RoboDK station: welding.rdk

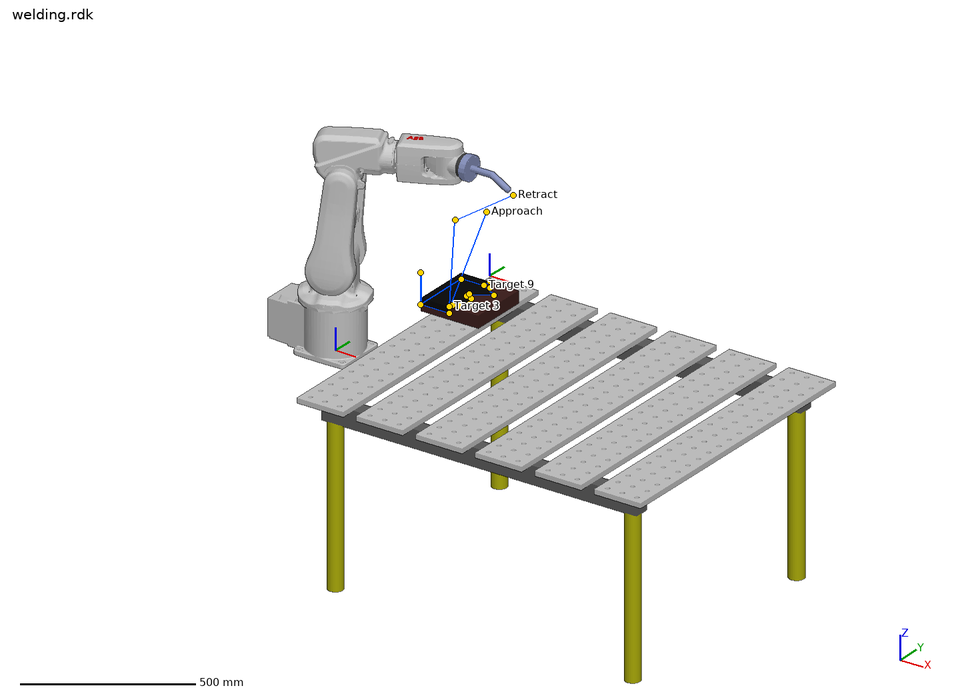
[picture v0: the station drawn from its stored meshes, robots at their saved joint values, targets as dots, program paths as lines]
Station welding (saved by RoboDK 5.3.4). Poses are relative to the parent item; angles as X-Y-Z fixed-axis rotations.
  - frame ABB IRB 120-3/0.6 Base at (0, 0, 0) mm
    - robot ABB IRB 120-3/0.6: 6 axes, payload 3 kg, reach 580 mm, repeatability 0.01 mm, weight 25 kg
        modified DH rows (alpha deg, a mm, theta deg, d mm): 0, 0, 0, 290; -90, 0, -90, 0; 0, 270, 0, 0; -90, 70, 0, 302; 90, 0, 0, 0; -90, 0, 180, 72
        joint limits [-165, -110, -90, -160, -120, -400] to [165, 110, 70, 160, 120, 400]; home [0, 0, 0, 0, 0, 0]; saved at [23.746, 6.012, -6.294, -89.359, 23.748, 89.3]
      - tool AssemblyWeldingTorch, TCP at (45, 0, 150) mm, rotated rx 0 ry 30 rz 0 deg, size 80 x 153.6 x 80.2 mm, geometry from AssemblyWeldingTorch.STEP
  - object Table at (800, 0, 100) mm, size 1193.8 x 965.2 x 609.6 mm, geometry from welding_table.sld
  - frame worktable at (200, 480, 100) mm
    - object Task1_Part2 at (180, -600, 200) mm, rotated rx 90 ry 0 rz 0 deg, size 160 x 20 x 200 mm, geometry from Task1_Part2.STEP
    - object Task1_Part1 at (280, -600, 200) mm, rotated rx 90 ry 0 rz 0 deg, size 200 x 40 x 200 mm, geometry from Task1_Part1.STEP
    - target Approach (Cartesian target) at (324, -480, 485) mm, rotated rx -180 ry 60 rz -180 deg; joints [0, 0, 0, 0, 0, 0] of ABB IRB 120-3/0.6
    - target Target 3 (Cartesian target) at (280, -600, 220) mm, rotated rx -180 ry 30 rz 180 deg; joints [-21.146, 7.513, 21.973, -96.878, -18.342, 86.297] of ABB IRB 120-3/0.6
    - target Target 4 (Cartesian target) at (280, -585, 220) mm, rotated rx -177.69 ry 30 rz 179.62 deg; joints [-17.055, 5.876, 23.812, 85.17, 12.458, -94.648] of ABB IRB 120-3/0.6
    - target Target 6 (Cartesian target) at (280, -515, 220) mm, rotated rx -177.69 ry 30 rz -175.38 deg; joints [-7.356, 3.4, 26.47, 86.971, 8.377, -94.106] of ABB IRB 120-3/0.6
    - target Target 7 (Cartesian target) at (280, -500, 220) mm, rotated rx -177.69 ry 20 rz -175.38 deg; joints [-3.841, 7.541, 16.793, 16.097, 16.374, -22.068] of ABB IRB 120-3/0.6
    - target Target 8 (Cartesian target) at (340, -465, 220) mm, rotated rx -177.69 ry 20 rz -175.38 deg; joints [1.761, 20.013, 1.699, 0.611, 18.24, -3.567] of ABB IRB 120-3/0.6
    - target Target 9 (Cartesian target) at (280, -430, 220) mm, rotated rx -177.69 ry 20 rz -175.38 deg; joints [7.944, 8.066, 16.204, -16.244, 16.455, 16.603] of ABB IRB 120-3/0.6
    - target Target 10 (Cartesian target) at (280, -400, 220) mm, rotated rx -177.69 ry 30 rz -175.38 deg; joints [13.586, 4.724, 25.061, -86.161, 9.774, 89.486] of ABB IRB 120-3/0.6
    - target Target 10-11 turning (Cartesian target) at (280, -400, 220) mm, rotated rx -90 ry 0 rz -150 deg; joints [36.548, 32.886, 19.556, 71.022, -75.96, 234.799] of ABB IRB 120-3/0.6
    - target Target 11 (Cartesian target) at (280, -400, 200) mm, rotated rx -90 ry 0 rz -150 deg; joints [36.548, 35.685, 19.831, 70.324, -76.978, -122.216] of ABB IRB 120-3/0.6
    - target Target 12 (Cartesian target) at (180, -400, 200) mm, rotated rx -90 ry 0 rz -150 deg; joints [47.566, 24.233, 38.454, -101.084, 84.33, 63.237] of ABB IRB 120-3/0.6
    - target Target 12-13 turning (Cartesian target) at (180, -400, 200) mm, rotated rx -90 ry 0 rz -60 deg; joints [-21.316, 14.165, 53.197, -81.976, -86.668, -67.596] of ABB IRB 120-3/0.6
    - target Target 13 (Cartesian target) at (180, -600, 200) mm, rotated rx -90 ry 0 rz -60 deg; joints [-51.555, 33.15, 24.081, -108.374, -101.47, -59.093] of ABB IRB 120-3/0.6
    - target Target 13-14 protect (Cartesian target) at (180, -600, 300) mm, rotated rx -90 ry 0 rz -60 deg; joints [-51.555, 20.557, 19.922, -104.383, -106.228, -42.541] of ABB IRB 120-3/0.6
    - target Target 13-14 turning (Cartesian target) at (180, -600, 200) mm, rotated rx 90 ry 0 rz 150 deg; joints [-52.09, 28.884, 31.081, 96.859, 86.05, -60.202] of ABB IRB 120-3/0.6
    - target Target 14 (Cartesian target) at (280, -600, 200) mm, rotated rx 90 ry 0 rz 150 deg; joints [-41.03, 39.706, 12.971, -74.711, -78.633, 125.792] of ABB IRB 120-3/0.6
    - target Target 15 (Cartesian target) at (280, -600, 220) mm, rotated rx 90 ry 0 rz 150 deg; joints [-41.03, 37.083, 12.697, 104.707, 77.883, -51.349] of ABB IRB 120-3/0.6
    - target protect (Cartesian target) at (300, -600, 500) mm, rotated rx 90 ry 0 rz 150 deg; joints [-39.266, 27.499, -27.594, 89.964, 69.266, 0.102] of ABB IRB 120-3/0.6
    - target Retract (Cartesian target) at (324, -347.14, 485) mm, rotated rx 180 ry 60 rz 180 deg; joints [23.746, 6.012, -6.294, -89.359, 23.748, 89.3] of ABB IRB 120-3/0.6
    - target Target 21 (Cartesian target) at (300.57, -578.32, 220) mm, rotated rx -180 ry 30 rz -180 deg; joints [-16.552, 10.076, 19.054, -97.54, -14.41, 89.33] of ABB IRB 120-3/0.6
    - target Target 22 (Cartesian target) at (315, -550, 220) mm, rotated rx -180 ry 30 rz -180 deg; joints [-11.462, 11.541, 17.34, -99.199, -10.04, 93.551] of ABB IRB 120-3/0.6
    - target Target 23 (Cartesian target) at (300.57, -521.68, 220) mm, rotated rx -180 ry 30 rz -180 deg; joints [-7.182, 7.675, 21.791, -96.672, -6.258, 93.106] of ABB IRB 120-3/0.6
    - target quidian (Cartesian target) at (280, -500, 220) mm, rotated rx -177.69 ry 30 rz -175.38 deg; joints [-4.616, 3.073, 26.813, 87.573, 6.003, -93.336] of ABB IRB 120-3/0.6
    - target 20-30reset (Cartesian target) at (280, -430, 220) mm, rotated rx -177.69 ry 30 rz -175.38 deg; joints [8.247, 3.54, 26.323, -87.432, 5.146, 88.089] of ABB IRB 120-3/0.6
  - program Prog1 (22 instructions, listed below)
  - program main (1 instructions, listed below)
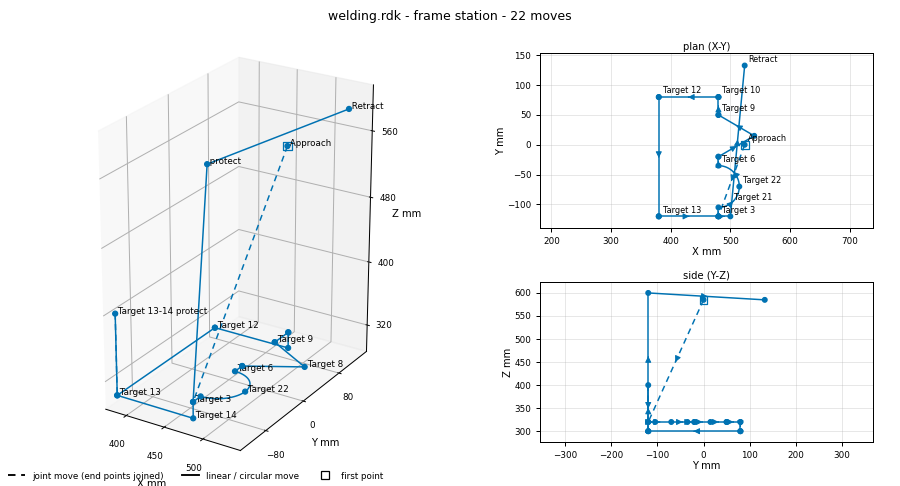
[picture p0: tool path of welding.rdk in frame station, 22 of 22 moves have a stored position in this frame; points joined in program order, loops and branches not executed]

--- program Prog1 (robot ABB IRB 120-3/0.6) ---
  MoveJ (Approach)
  MoveJ (Target 3)
  MoveL (Target 4)
  MoveC (Target 21, Target 22)
  MoveC (Target 23, Target 6)
  MoveL (quidian)
  MoveJ (Target 7)
  MoveL (Target 8)
  MoveL (Target 9)
  MoveJ (20-30reset)
  MoveL (Target 10)
  MoveL (Target 10-11 turning)
  MoveL (Target 11)
  MoveL (Target 12)
  MoveJ (Target 12-13 turning)
  MoveL (Target 13)
  MoveL (Target 13-14 protect)
  MoveJ (Target 13-14 turning)
  MoveL (Target 14)
  MoveL (Target 15)
  MoveL (protect)
  MoveL (Retract)

--- program main (robot ABB IRB 120-3/0.6) ---
  调用 Prog1
